{attribute 'enable_dynamic_creation'}	
{attribute 'no_explicit_call' := 'do not call this function block directly'} 
FUNCTION_BLOCK ArgumentOutOfRangeException EXTENDS GeneralException
VAR
	_ClassName : STRING := __POUNAME();
END_VAR

{attribute 'monitoring' := 'call'}
PROPERTY ClassName : STRING
GET
ClassName := _ClassName;
END_GET
END_PROPERTY

METHOD Clone : IObject
VAR
	exceptionClone : POINTER TO ArgumentOutOfRangeException;
END_VAR
exceptionClone := __NEW(ArgumentOutOfRangeException);

Clone := InternalClone(exceptionClone);
END_METHOD

METHOD Throw
VAR_INPUT
	sourceNamespaceName : STRING;
	sourceClassName : STRING;
	sourceMethodName : STRING;
	sourcePosition : STRING;
	argumentName : STRING;
	argumentValue : ANY;
	fatal : BOOL := FALSE;
END_VAR
VAR
	valueAsString : WSTRING(255);
	stringBuilder : WideStringBuilder;
	message : ERROR_MESSAGE;
	zeroErrorCode : UDINT;
	nullInnerException : REFERENCE TO Exception REF= 0;
END_VAR
valueAsString := WideStringHelper.InternalAnyToString(argumentValue);

stringBuilder
	.AppendString("Argument '")
	.Append(argumentName)
	.AppendString("' has invalid value '")
	.AppendString(valueAsString)
	.AppendString("in method or function '");

AppendProgramOrganizationUnitFullName(stringBuilder);

stringBuilder
	.AppendString("'")
	.AssignToString(message);

InternalThrow(sourceNamespaceName, sourceClassName, sourceMethodName, sourcePosition, message, zeroErrorCode, fatal, nullInnerException);
END_METHOD

END_FUNCTION_BLOCK

(* stored: Version 1.1.0.1
   POU ArgumentOutOfRangeException: Id {98d20286-f8bd-41e5-8b87-fcb4b5d7ca5e}, SpecialFunc None
   Property ClassName: Id {c27874b7-4abc-48c2-950c-b0bb5f01f34d}
   Get Get: Id {731dacbe-6b4c-4a54-a726-b999af608436}
   Method Clone: Id {6b5d2ab8-4da4-4d0d-bf7c-087be7ca447f}
   Method Throw: Id {5feec76b-4654-49c9-b2bc-8cf052990d28} *)
